FUNCTION_BLOCK Boia (* Composite Function Block Type *)
  (* Standard: 61499-2 *)
  (* Version 0.0, 2/9/2026, Schneider Electric, template *)
  PACKAGE Hidryco.HidrycoLib;
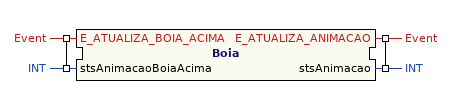
  EVENT_INPUT
    E_ATUALIZA_BOIA_ACIMA WITH stsAnimacaoBoiaAcima;
  END_EVENT
  EVENT_OUTPUT
    E_ATUALIZA_ANIMACAO WITH stsAnimacao;
  END_EVENT
  VAR_INPUT
    stsAnimacaoBoiaAcima : INT;
  END_VAR
  VAR_OUTPUT
    stsAnimacao : INT;
  END_VAR
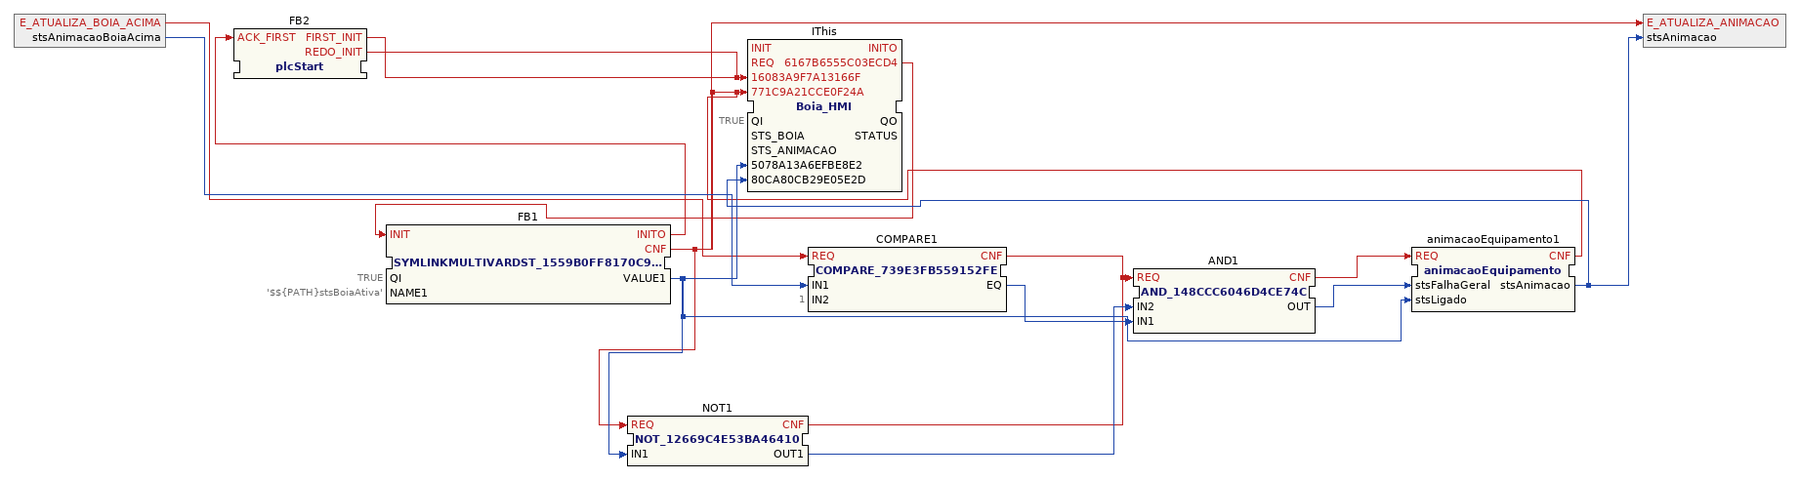
  FBS
    FB1 : SYMLINKMULTIVARDST_1559B0FF8170C9BA0(QI := TRUE, NAME1 := '$${PATH}stsBoiaAtiva'); {SET_ATTRIBUTE(Configuration.GenericFBType.InterfaceParams, Runtime.System#I:=1;VALUE${I$}:BOOL)}
    FB2 : plcStart;
    IThis : Boia_HMI(QI := TRUE);
    AND1 : AND_148CCC6046D4CE74C; {SET_ATTRIBUTE(Configuration.GenericFBType.InterfaceParams, Runtime.Standard#CNT:=2)}
    animacaoEquipamento1 : animacaoEquipamento;
    NOT1 : NOT_12669C4E53BA46410; {SET_ATTRIBUTE(Configuration.GenericFBType.InterfaceParams, Runtime.Standard#CNT:=1)}
    COMPARE1 : COMPARE_739E3FB559152FE(IN2 := 1); {SET_ATTRIBUTE(Configuration.GenericFBType.InterfaceParams, Runtime.Standard#CNT:=2;IN${CNT$}:INT)}
  END_FBS
  EVENT_CONNECTIONS
    FB1.INITO TO FB2.ACK_FIRST;
    FB1.CNF TO E_ATUALIZA_ANIMACAO;
    FB1.CNF TO NOT1.REQ;
    NOT1.CNF TO AND1.REQ;
    AND1.CNF TO animacaoEquipamento1.REQ;
    FB2.FIRST_INIT TO IThis.16083A9F7A13166F;
    FB2.REDO_INIT TO IThis.16083A9F7A13166F;
    FB1.CNF TO IThis.771C9A21CCE0F24A;
    animacaoEquipamento1.CNF TO IThis.771C9A21CCE0F24A;
    IThis.6167B6555C03ECD4 TO FB1.INIT;
    E_ATUALIZA_BOIA_ACIMA TO COMPARE1.REQ;
    COMPARE1.CNF TO AND1.REQ;
  END_CONNECTIONS
  DATA_CONNECTIONS
    FB1.VALUE1 TO NOT1.IN1;
    NOT1.OUT1 TO AND1.IN2;
    AND1.OUT TO animacaoEquipamento1.stsFalhaGeral;
    FB1.VALUE1 TO animacaoEquipamento1.stsLigado;
    FB1.VALUE1 TO IThis.5078A13A6EFBE8E2;
    animacaoEquipamento1.stsAnimacao TO IThis.80CA80CB29E05E2D;
    stsAnimacaoBoiaAcima TO COMPARE1.IN1;
    COMPARE1.EQ TO AND1.IN1;
    animacaoEquipamento1.stsAnimacao TO stsAnimacao;
  END_CONNECTIONS
END_FUNCTION_BLOCK
